FUNCTION_BLOCK Directory
VAR
	creator : FB_CreateDir; // can only create on level of folder
	remover : FB_RemoveDir; // can only remove topmost folder. Not folder with folders.

	listDir : FB_EnumFindFileList;	
	listingFinishedTrigger : F_TRIG;
	fileListDone : BOOL;
	checkingFolder : BOOL;
	checkingFileExistence : BOOL;

	page : ARRAY[0..50 - 1] OF ST_FindFileEntry;
	_FileNameList : ARRAY[0..50 - 1] OF T_MaxString;
	_FileExists : BOOL;
END_VAR
VAR CONSTANT
	EntriesPerPage : INT := 50;
END_VAR

METHOD PRIVATE Abort
VAR_INPUT
END_VAR
listDir(
	bExecute := TRUE,
	eCmd := E_EnumCmdType.eEnumCmd_Abort
);
listDir(bExecute := FALSE);
END_METHOD

{attribute 'TcRpcEnable':='1'}
METHOD Create
VAR_INPUT
	path : T_MaxString;
END_VAR
creator(
	sPathName := path,
	bExecute := TRUE,
);
END_METHOD

METHOD Cyclic
VAR
	i : INT;
END_VAR
creator(bExecute := FALSE);
remover(bExecute := FALSE);

listDir(
	pFindList := ADR(page),
	cbFindList := SIZEOF(page)
);

listingFinishedTrigger(CLK := listDir.bBusy);
IF (listingFinishedTrigger.Q AND listDir.eCmd <> E_EnumCmdType.eEnumCmd_Abort) THEN

	listDir(bExecute := FALSE);
	fileListDone := TRUE;
	
	FOR i := 0 TO EntriesPerPage - 1 DO
		_FileNameList[i] := page[i].sFileName;
		
		IF (checkingFileExistence) THEN
			IF (page[i].fileAttributes.bDirectory = checkingFolder
				AND page[i].sFileName <> '') THEN
				_FileExists := TRUE;
			END_IF
		END_IF
	END_FOR
	
	IF (NOT listDir.bEOE) THEN
		Abort();
	END_IF
END_IF
END_METHOD

{attribute 'monitoring' := 'call'}
PROPERTY FileExists : BOOL
GET
FileExists := _FileExists;
END_GET
END_PROPERTY

{attribute 'monitoring' := 'call'}
PROPERTY FileNameList : REFERENCE TO ARRAY[0..49] OF T_MaxString
GET
FileNameList REF= _FileNameList;
END_GET
END_PROPERTY

METHOD CheckFileExists
VAR_INPUT
	path : T_MaxString;
	folder : BOOL; // FALSE = File, TRUE = Folder
END_VAR
IF (NOT listDir.bBusy) THEN
	
	List(path);
	
	_FileExists := FALSE;
	checkingFileExistence := TRUE;
	checkingFolder := folder;
END_IF
END_METHOD

 // Usage of * wildcard recommended
 // Add * to the end of path to list all files
METHOD List
VAR_INPUT
	path : T_MaxString;
END_VAR
IF (NOT listDir.bBusy) THEN
	
	checkingFileExistence := FALSE;
	fileListDone := FALSE;
	
	listDir(bExecute := FALSE);
	listDir(
		sPathName := path,
		eCmd := E_EnumCmdType.eEnumCmd_First,
		bExecute := TRUE
	);
END_IF
END_METHOD

METHOD Remove
VAR_INPUT
	path : T_MaxString;
END_VAR
remover(
	sPathName := path,
	bExecute := TRUE,
);
END_METHOD

END_FUNCTION_BLOCK

(* stored: Version 1.1.0.1, ProductVersion 3.1.4024.12
   POU Directory: Id {2249bebd-97d6-0598-2285-3e82d8824005}, SpecialFunc None
   Method Abort: Id {3028eaae-44eb-0639-284d-cd8671b65d39}
   Method Create: Id {5261a63a-4bf4-05eb-3d54-5f8d5f5f5b50}
   Method Cyclic: Id {f3d38fcf-5c78-0bd2-0f7f-a8d48fb4188d}
   Property FileExists: Id {90ece582-5e1b-01dc-0274-516d568d103f}
   Get Get: Id {888b3ecc-224e-074c-06f8-8ccb5c9ed7a8}
   Property FileNameList: Id {8d6fa6ed-c4df-048c-3f37-69a9a0b7b188}
   Get Get: Id {4c8de85d-3a9d-0dc1-2bf7-958db259dc14}
   Method CheckFileExists: Id {153a5eb4-6f1b-0815-21fc-1d24e1d857f2}
   Method List: Id {3d045257-9a2c-01d9-167a-bfeb0b1760e1}
   Method Remove: Id {1bc872e8-0a59-0cee-2768-74b2c8c4a37c} *)
